ABB RobotStudio station: ProyectoRob.rsstnx

Station ProyectoRob (saved by RobotStudio 25.1.11167.1)
Controller IRB140_6_81
  mechanical unit ROB_1: IRB140_6_81_C_03, 6 joints, base frame (0, 0, 0) mm
Layout (positions relative to the parent item):
  - IRB140_6_81_C_03 [mechanism, from %ABB.RobotStudio.Models.IRB140%\IRB140_6_81_C_G_03.rslib] at (0, 0, 0) mm; joint values [0.2784, 0.4347, 0.5017, -3.1414, 0.9363, 1.5706] (rad or m)
  - SmartComponent_1 [smart component] at (472.11, 134.91, 531.5) mm, rotated rx -90 ry 0 rz -74.06 deg
      signals: DI DI_Open, DI DI_Close, DI DI_Att, DI DI_Dett
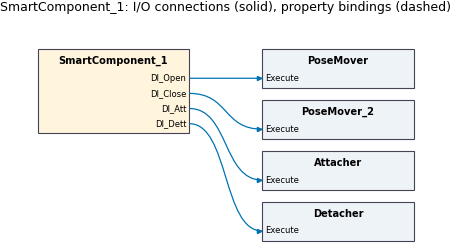
      connections:
        SmartComponent_1.DI_Open -> PoseMover.Execute
        SmartComponent_1.DI_Close -> PoseMover_2.Execute
        SmartComponent_1.DI_Att -> Attacher.Execute
        SmartComponent_1.DI_Dett -> Detacher.Execute
    - PoseMover [smart component, from Components\PoseMover.rslib]
        properties: Mechanism=Griper; Pose=2; Duration=1
    - PoseMover_2 [smart component, from Components\PoseMover.rslib]
        properties: Mechanism=Griper; Pose=1; Duration=1
    - Griper [mechanism] at (0, 0, 0) mm; joint values [-0.3491, 0.3491, 0, 0] (rad or m)
        TCP Griper_1 at (0, 17.5, 237) mm
        links: L1, L2, L3, L4, L5
    - Attacher [smart component, from Components\Attacher.rslib]
        properties: Parent=Detacher; Flange=0; Child=C10_2; Mount=false; Offset=[0 0 0]; Orientation=[0 0 0]
    - Detacher [smart component, from Components\Detacher.rslib]
        properties: Child=C10_2; KeepPosition=true
  - Band [part] at (0, -730, 440) mm, rotated rx 180 ry 0 rz 90 deg, size 200 x 800 x 460 mm
  - Est_2 [part] at (590, 375, 260) mm, rotated rx 180 ry 0 rz 0 deg, size 320 x 750 x 260 mm
  - C10_2 [part] at (700, 200, 260) mm, rotated rx 180 ry 0 rz 180 deg, size 69.9 x 70 x 20 mm
Attachment: SmartComponent_1 is attached to IRB140_6_81_C_03 / Link6
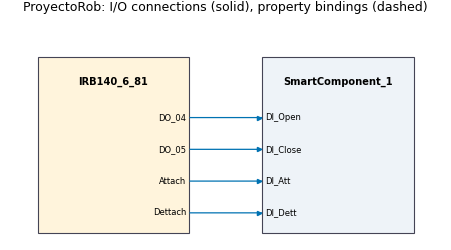
Station logic (signal -> signal, property => property):
  IRB140_6_81.DO_04 -> SmartComponent_1.DI_Open
  IRB140_6_81.DO_05 -> SmartComponent_1.DI_Close
  IRB140_6_81.Attach -> SmartComponent_1.DI_Att
  IRB140_6_81.Dettach -> SmartComponent_1.DI_Dett
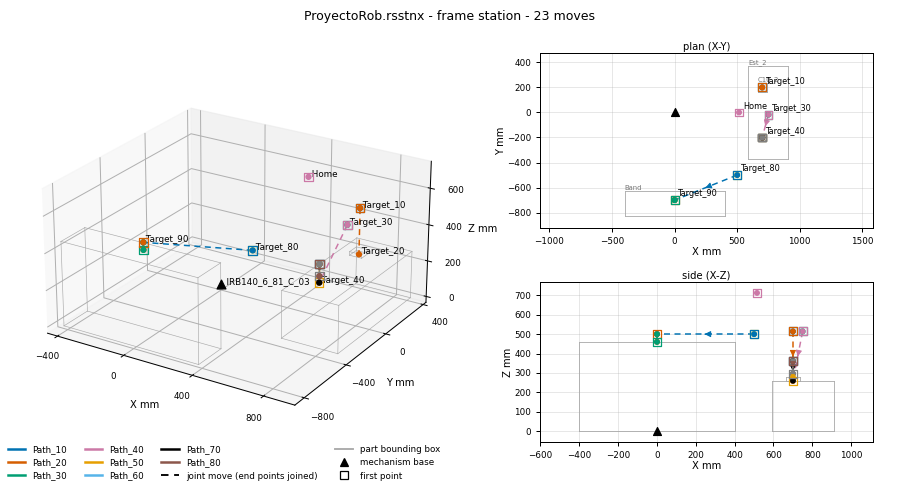
[picture p0: tool path of ProyectoRob.rsstnx in frame station, 23 of 23 moves have a stored position in this frame; points joined in program order, loops and branches not executed]
Targets, tools, work objects and paths stored in the station, written as RAPID:
! task T_ROB1
MODULE CalibData
  PERS tooldata Griper:=[TRUE,[[0,17.5,237],[0.5,-0.5,0.5,0.5]],[1,[0,17.5,237],[1,0,0,0],1,1,1]];
  TASK PERS wobjdata Mesa:=[FALSE,TRUE,"",[[590,375,260],[0,0,1,0]],[[0,0,0],[1,0,0,0]]];
ENDMODULE

! task T_ROB1
MODULE Module1
  CONST robtarget Target_10:=[[-110,-175,-254],[0.990340804,0,0,-0.138654579],[0,-2,0,0],[9E+09,9E+09,9E+09,9E+09,9E+09,9E+09]];
  CONST robtarget Target_20:=[[-110,-175,0],[0.990340804,0,0,-0.138654579],[0,0,0,0],[9E+09,9E+09,9E+09,9E+09,9E+09,9E+09]];
  CONST robtarget Target_30:=[[-160,-392.5,-253.927],[1,0,0,0],[0,0,0,0],[9E+09,9E+09,9E+09,9E+09,9E+09,9E+09]];
  CONST robtarget Target_40:=[[-110,-575,0],[0.990340804,0,0,0.138654579],[0,0,0,0],[9E+09,9E+09,9E+09,9E+09,9E+09,9E+09]];
  CONST robtarget Target_50:=[[-110,-575,-100],[0.990340804,0,0,0.138654579],[0,0,0,0],[9E+09,9E+09,9E+09,9E+09,9E+09,9E+09]];
  CONST robtarget Target_60:=[[-110,-575,-100],[0,0.990340804,0.138654579,0],[0,0,0,0],[9E+09,9E+09,9E+09,9E+09,9E+09,9E+09]];
  CONST robtarget Target_70:=[[-110,-575,-35],[0,0.990340804,0.138654579,0],[0,0,0,0],[9E+09,9E+09,9E+09,9E+09,9E+09,9E+09]];
  CONST robtarget Target_80:=[[90,-875,-240],[0.923879533,0,0,0.382683432],[0,0,0,0],[9E+09,9E+09,9E+09,9E+09,9E+09,9E+09]];
  CONST robtarget Target_90:=[[590,-1075,-240],[0.707106781,0,0,0.707106781],[0,0,0,0],[9E+09,9E+09,9E+09,9E+09,9E+09,9E+09]];
  CONST robtarget Target_100:=[[590,-1075,-200],[0.707106781,0,0,0.707106781],[0,0,0,0],[9E+09,9E+09,9E+09,9E+09,9E+09,9E+09]];
  CONST robtarget Home:=[[515,0,712],[0.707106781,0,0.707106781,0],[0,0,0,0],[9E+09,9E+09,9E+09,9E+09,9E+09,9E+09]];
  PROC main()
    Path_140;
    Set DO_01;
    Path_10;
    Set DO_04;
    Reset DO_04;
    WaitTime 1;
    Path_20;
    WaitTime 1;
    Set DO_05;
    Reset DO_05;
    Set Attach;
    Reset Attach;
    WaitTime 1;
    Path_10;
    Path_30;
    Path_40;
    WaitTime 1;
    Set DO_04;
    Reset DO_04;
    WaitTime 1;
    Set Dettach;
    Reset Dettach;
    Path_50;
    WaitTime 10;
    Path_70;
    WaitTime 1;
    Set DO_05;
    Reset DO_05;
    WaitTime 2;
    Set Attach;
    Reset Attach;
    Path_50;
    Path_60;
    Path_80;
    WaitTime 1;
    Set DO_04;
    Reset DO_04;
    WaitTime 1;
    Set Dettach;
    Reset Dettach;
    Path_90;
    WaitTime 10;
    Path_80;
    WaitTime 2;
    Set DO_05;
    Reset DO_05;
    Set Attach;
    Reset Attach;
    WaitTime 1;
    Path_100;
    Path_110;
    Path_120;
    WaitTime 1;
    Set DO_04;
    Reset DO_04;
    WaitTime 1;
    Set Dettach;
    Reset Dettach;
    Path_130;
    WaitTime 1;
    Set DO_05;
    Reset DO_05;
    Path_100;
    Path_30;
    Reset DO_01;
  ENDPROC
  PROC Path_10()
    MoveJ Target_10,v100,z10,Griper\WObj:=Mesa;
  ENDPROC
  PROC Path_20()
    MoveJ Target_10,v100,z10,Griper\WObj:=Mesa;
    MoveJ Target_20,v100,z10,Griper\WObj:=Mesa;
  ENDPROC
  PROC Path_30()
    MoveJ Target_30,v100,z10,Griper\WObj:=Mesa;
  ENDPROC
  PROC Path_40()
    MoveJ Target_30,v100,z10,Griper\WObj:=Mesa;
    MoveJ Target_40,v100,z10,Griper\WObj:=Mesa;
  ENDPROC
  PROC Path_50()
    MoveJ Target_40,v100,z10,Griper\WObj:=Mesa;
    MoveJ Target_50,v100,z10,Griper\WObj:=Mesa;
  ENDPROC
  PROC Path_60()
    MoveJ Target_60,v100,z100,Griper\WObj:=Mesa;
  ENDPROC
  PROC Path_70()
    MoveJ Target_50,v100,z10,Griper\WObj:=Mesa;
    MoveJ Target_40,v100,z10,Griper\WObj:=Mesa;
  ENDPROC
  PROC Path_80()
    MoveJ Target_60,v100,z10,Griper\WObj:=Mesa;
    MoveJ Target_70,v100,z10,Griper\WObj:=Mesa;
  ENDPROC
  PROC Path_90()
    MoveJ Target_70,v100,z10,Griper\WObj:=Mesa;
    MoveJ Target_60,v100,z10,Griper\WObj:=Mesa;
  ENDPROC
  PROC Path_100()
    MoveJ Target_80,v100,z10,Griper\WObj:=Mesa;
  ENDPROC
  PROC Path_110()
    MoveJ Target_80,v100,z10,Griper\WObj:=Mesa;
    MoveJ Target_90,v100,z10,Griper\WObj:=Mesa;
  ENDPROC
  PROC Path_120()
    MoveJ Target_90,v100,z10,Griper\WObj:=Mesa;
    MoveJ Target_100,v100,z10,Griper\WObj:=Mesa;
  ENDPROC
  PROC Path_130()
    MoveJ Target_100,v100,z10,Griper\WObj:=Mesa;
    MoveJ Target_90,v100,z10,Griper\WObj:=Mesa;
  ENDPROC
  PROC Path_140()
    MoveJ Home,v1000,z100,tool0\WObj:=wobj0;
  ENDPROC
ENDMODULE

